{attribute 'qualified_only'}
{attribute 'analysis' := '-33'}
VAR_GLOBAL
	MonitorTestData		: MonitorTest;
	ReadTestData		: ReadTest;
	SymbolTestData		: SymbolTest;
	WriteTestData		: WriteTest;
END_VAR

(* stored: Version 1.1.0.1, ProductVersion 3.1.4024.12
   GVL AdsNet7: Id {58c6384f-95cc-00d6-0aa6-a8eb1ce8870c} *)
